PROGRAM lightControl
VAR
    userNearMirror : BOOL;  // Variable to store whether the user is near the mirror
END_VAR

// Call the function to check if the user is near the mirror
userNearMirror := checkDistance(distance_in_function := GVL.distance);

// Turn on the light if the user is near the mirror
IF userNearMirror = TRUE THEN
    GVL.lightStatus := TRUE;
ELSIF userNearMirror = FALSE THEN
    // Start the timer when the user moves away from the mirror
    timerControl();  
END_IF

END_PROGRAM

(* stored: Version 1.1.0.1, ProductVersion 3.1.4024.12
   POU lightControl: Id {0edb4d64-9ccb-48ce-8cde-93a1666a05b9}, SpecialFunc None *)
